TYPE ST_AutoMode_ShippingRobot_MoveAbs :
STRUCT
	Command 	: ST_CommandBasic;
	Status 		: ST_StatusBasic;
	Info 		: ST_RobotRegionMove_Info;
	bCompleteRequest 	: BOOL;
	bTransCVInPosition	: BOOL;
END_STRUCT
END_TYPE

(* stored: Version 1.1.0.1, ProductVersion 3.1.4024.13
   DUT ST_AutoMode_ShippingRobot_MoveAbs: Id {fc799fca-a312-4096-b069-4e161397a5a4} *)
